Staubli VAL3: setupRosMsgs.pgx

public program setupRosMsgs()
begin
  // Copyright (c) 2016, Ocado Technology - Robotics Research Team
  //
  // Licensed under the Apache License, Version 2.0 (the "License");
  // you may not use this file except in compliance with the License.
  // You may obtain a copy of the License at
  //
  //     http://www.apache.org/licenses/LICENSE-2.0
  //
  // Unless required by applicable law or agreed to in writing, software
  // distributed under the License is distributed on an "AS IS" BASIS,
  // WITHOUT WARRANTIES OR CONDITIONS OF ANY KIND, either express or implied.
  // See the License for the specific language governing permissions and
  // limitations under the License.



  // Joint state message (ID 10)
  // prefix length = 12 + 44
  rosJointMsg.prefix.nLength=56
  rosJointMsg.header.nMsgType=10
  rosJointMsg.header.nCommType=1
  rosJointMsg.header.nReplyCode=0
  // sequence
  rosJointMsg.jointState.nSeq=0



  // Joint trajectory point message (ID 11)
  // prefix length = 12 + 52
  rosTrajPtAck.prefix.nLength=64
  rosTrajPtAck.header.nMsgType=11
  rosTrajPtAck.header.nCommType=3
  // reply: 1 = success, 2 = failure
  rosTrajPtAck.header.nReplyCode=1
  // joints are assumed to be initiliased to zero

  // the message bellow will be filled upon reception
  rosTrajPtMsg.prefix.nLength=64



  // Robot status message (ID 13)
  // prefix length = 12 + 28
  rosStatusMsg.prefix.nLength=40
  rosStatusMsg.header.nMsgType=13
  rosStatusMsg.header.nCommType=1
  rosStatusMsg.header.nReplyCode=0



  // Joint trajectory point full message (ID 14)
  // prefix length = 12 + 136
  rosTrajPtFAck.prefix.nLength=148
  rosTrajPtFAck.header.nMsgType=14
  rosTrajPtFAck.header.nCommType=3
  // reply: 1 = success, 2 = failure
  rosTrajPtFAck.header.nReplyCode=1
  // body (data) assumed to be initialised to zero

  // the message bellow will be filled upon reception
  rosTrajPtFMsg.prefix.nLength=148

  // Cartesian trajectory point message (ID 31)
  // prefix length = 12 + 48
  rosTrajPtCartesianAck.prefix.nLength=60
  rosTrajPtCartesianAck.header.nMsgType=31
  rosTrajPtCartesianAck.header.nCommType=3
  // reply: 1 = success, 2 = failure
  rosTrajPtCartesianAck.header.nReplyCode=1
  // position, orientation, velocities, etc are assumed to be initiliased to zero

  // the message bellow will be filled upon reception
  rosTrajPtCartesianMsg.prefix.nLength=60


  // Joint feedback message (ID 15)
  // prefix length = 12 + 132
  rosJointFbkMsg.prefix.nLength=144
  rosJointFbkMsg.header.nMsgType=15
  rosJointFbkMsg.header.nCommType=1
  rosJointFbkMsg.header.nReplyCode=0
end
